// TIA Portal V18 export
DATA_BLOCK "Main_Safety_RTG1_DB"   // DB1, F_DB
{ DB_Accessible_From_OPC_UA := 'FALSE' }
NAME : FUSI
// stored: DBAccessibleFromOPCUA false, InstanceOfName Main_Safety_RTG1, InstanceOfType FB
"Main_Safety_RTG1"
BEGIN
END_DATA_BLOCK
